// TIA Portal V17 export
// export: Created 2023-09-01T12:47:09.6374792Z, ExportSetting WithDefaults, DisplayName Totally Integrated Automation Portal, DisplayVersion V17 Update 6, DisplayName TIA Portal Openness, DisplayVersion V17 Update 6, DisplayName TIA Portal Teamcenter Gateway, DisplayVersion V17 Update 6, DisplayName TIA Portal Version Control Interface, DisplayVersion V17, DisplayName Simotion SCOUT TIA, DisplayVersion 5.4.3.0, DisplayName TIA Portal Test Suite Advanced, DisplayVersion V17 Update 1, DisplayName SIMOCODE ES, DisplayVersion V17 Update 5, DisplayName SINAMICS Startdrive Advanced, DisplayVersion V17 SP1, DisplayName SINAMICS Startdrive G130, G150, S120, S150, SINAMICS MV, S210, DisplayVersion V17 SP1, DisplayName SINAMICS Startdrive G110M, G120, G120C, G120D, G120P, G115D, DisplayVersion V17 SP1, DisplayName SIRIUS Safety ES, DisplayVersion V17 Update 5, DisplayName STEP 7 Professional, DisplayVersion V17 Update 6, DisplayName STEP 7 CFC, DisplayVersion V17 Update 1, DisplayName STEP 7 Safety, DisplayVersion V17 Update 6, DisplayName WinCC Advanced, DisplayVersion V17 Update 6, DisplayName SIMATIC Visualization Architect, DisplayVersion V17 Update 5
FUNCTION "06_Feedback Error" : Void   // FC7, F_LAD
TITLE = Mirror F_FDBACK.ERROR
{ S7_Optimized_Access := 'TRUE' }
VERSION : 0.1
// stored: AutoNumber true, IsIECCheckEnabled false, UDAEnableTagReadback false
BEGIN

REGION Network 1: !!COLUMN_1$$
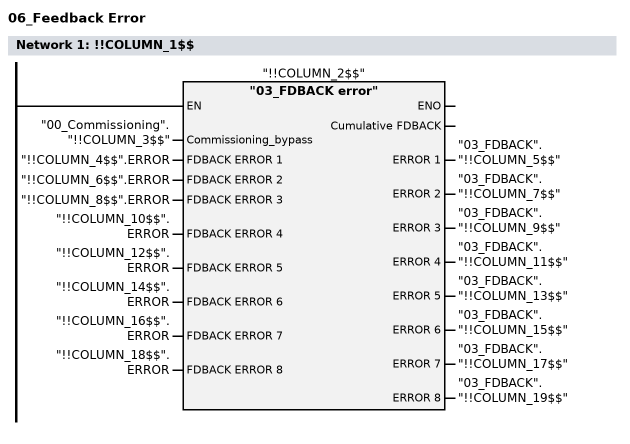
   RUNG wire#powerrail
      "!!COLUMN_2$$"(Commissioning_bypass := "00_Commissioning"."!!COLUMN_3$$", "FDBACK ERROR 1" := "!!COLUMN_4$$".ERROR, "FDBACK ERROR 2" := "!!COLUMN_6$$".ERROR, "FDBACK ERROR 3" := "!!COLUMN_8$$".ERROR, "FDBACK ERROR 4" := "!!COLUMN_10$$".ERROR, "FDBACK ERROR 5" := "!!COLUMN_12$$".ERROR, "FDBACK ERROR 6" := "!!COLUMN_14$$".ERROR, "FDBACK ERROR 7" := "!!COLUMN_16$$".ERROR, "FDBACK ERROR 8" := "!!COLUMN_18$$".ERROR, "Cumulative FDBACK" =>, "ERROR 1" => "03_FDBACK"."!!COLUMN_5$$", "ERROR 2" => "03_FDBACK"."!!COLUMN_7$$", "ERROR 3" => "03_FDBACK"."!!COLUMN_9$$", "ERROR 4" => "03_FDBACK"."!!COLUMN_11$$", "ERROR 5" => "03_FDBACK"."!!COLUMN_13$$", "ERROR 6" => "03_FDBACK"."!!COLUMN_15$$", "ERROR 7" => "03_FDBACK"."!!COLUMN_17$$", "ERROR 8" => "03_FDBACK"."!!COLUMN_19$$")
   END_RUNG
   // the same network as SCL:
   "!!COLUMN_2$$"(Commissioning_bypass := "00_Commissioning"."!!COLUMN_3$$",   // "03_FDBACK error"
                  "FDBACK ERROR 1" := "!!COLUMN_4$$".ERROR,
                  "FDBACK ERROR 2" := "!!COLUMN_6$$".ERROR,
                  "FDBACK ERROR 3" := "!!COLUMN_8$$".ERROR,
                  "FDBACK ERROR 4" := "!!COLUMN_10$$".ERROR,
                  "FDBACK ERROR 5" := "!!COLUMN_12$$".ERROR,
                  "FDBACK ERROR 6" := "!!COLUMN_14$$".ERROR,
                  "FDBACK ERROR 7" := "!!COLUMN_16$$".ERROR,
                  "FDBACK ERROR 8" := "!!COLUMN_18$$".ERROR,
                  "ERROR 1" => "03_FDBACK"."!!COLUMN_5$$",
                  "ERROR 2" => "03_FDBACK"."!!COLUMN_7$$",
                  "ERROR 3" => "03_FDBACK"."!!COLUMN_9$$",
                  "ERROR 4" => "03_FDBACK"."!!COLUMN_11$$",
                  "ERROR 5" => "03_FDBACK"."!!COLUMN_13$$",
                  "ERROR 6" => "03_FDBACK"."!!COLUMN_15$$",
                  "ERROR 7" => "03_FDBACK"."!!COLUMN_17$$",
                  "ERROR 8" => "03_FDBACK"."!!COLUMN_19$$");
END_REGION
END_FUNCTION
